FUNCTION TryConvert_ULINT_TO_STRING : BOOL
VAR_INPUT
	in : ULINT;
	out : REFERENCE TO STRING;
END_VAR

out := ULINT_TO_STRING(in);
TryConvert_ULINT_TO_STRING := TRUE;

END_FUNCTION

(* stored: Version 1.1.0.1, ProductVersion 3.1.4024.12
   POU TryConvert_ULINT_TO_STRING: Id {50e61dd2-ba33-4f02-b42d-bc5b24e9ddd7}, SpecialFunc None *)
